// TIA Portal V20 export
TYPE "type_emRelations_em7_sequence"
// stored: Access Published, Namespace Unit1
   STRUCT
      Spare1 { S7_SetPoint := 'True'} : "LER_typeSequenceRelation";
      Spare2 { S7_SetPoint := 'True'} : "LER_typeSequenceRelation";
      Spare3 { S7_SetPoint := 'True'} : "LER_typeSequenceRelation";
      Spare4 { S7_SetPoint := 'True'} : "LER_typeSequenceRelation";
      Spare5 { S7_SetPoint := 'True'} : "LER_typeSequenceRelation";
      Spare6 { S7_SetPoint := 'True'} : "LER_typeSequenceRelation";
      Spare7 { S7_SetPoint := 'True'} : "LER_typeSequenceRelation";
      Spare8 { S7_SetPoint := 'True'} : "LER_typeSequenceRelation";
      Spare9 { S7_SetPoint := 'True'} : "LER_typeSequenceRelation";
   END_STRUCT;
END_TYPE
